PROGRAM Programma_2
VAR
    currentPlayer: BOOL;  // Bepaalt welke speler aan de beurt is
	zetGedaan: BOOL;
END_VAR

// Task 2: Speler zet zijn figuur
IF GVL.game_status = 1 THEN
    zetGedaan := FALSE; // Variabele om bij te houden of er een zet is gedaan

    // Bepaal welke speler aan de beurt is
    IF GVL.Player_1 THEN
        currentPlayer := TRUE;   // Speler 1 is actief
    ELSE
        currentPlayer := FALSE;  // Speler 2 is actief
    END_IF

    // Controleer of een rechthoek is geselecteerd en of deze leeg is
    // Als de rechthoek leeg is, vul het met het figuur van de speler
    IF GVL.Rechthoek_1 AND NOT (GVL.Driehoek_1 OR GVL.Rondje_1) THEN
        IF currentPlayer THEN
            GVL.Driehoek_1 := TRUE;  // Zet driehoek van speler 1
        ELSE
            GVL.Rondje_1 := TRUE;    // Zet rondje van speler 2
        END_IF
        zetGedaan := TRUE;
    ELSIF GVL.Rechthoek_2 AND NOT (GVL.Driehoek_2 OR GVL.Rondje_2) THEN
        IF currentPlayer THEN
            GVL.Driehoek_2 := TRUE;  // Zet driehoek van speler 1
        ELSE
            GVL.Rondje_2 := TRUE;    // Zet rondje van speler 2
        END_IF
        zetGedaan := TRUE;
    ELSIF GVL.Rechthoek_3 AND NOT (GVL.Driehoek_3 OR GVL.Rondje_3) THEN
        IF currentPlayer THEN
            GVL.Driehoek_3 := TRUE;  // Zet driehoek van speler 1
        ELSE
            GVL.Rondje_3 := TRUE;    // Zet rondje van speler 2
        END_IF
        zetGedaan := TRUE;
    ELSIF GVL.Rechthoek_4 AND NOT (GVL.Driehoek_4 OR GVL.Rondje_4) THEN
        IF currentPlayer THEN
            GVL.Driehoek_4 := TRUE;  // Zet driehoek van speler 1
        ELSE
            GVL.Rondje_4 := TRUE;    // Zet rondje van speler 2
        END_IF
        zetGedaan := TRUE;
    ELSIF GVL.Rechthoek_5 AND NOT (GVL.Driehoek_5 OR GVL.Rondje_5) THEN
        IF currentPlayer THEN
            GVL.Driehoek_5 := TRUE;  // Zet driehoek van speler 1
        ELSE
            GVL.Rondje_5 := TRUE;    // Zet rondje van speler 2
        END_IF
        zetGedaan := TRUE;
    ELSIF GVL.Rechthoek_6 AND NOT (GVL.Driehoek_6 OR GVL.Rondje_6) THEN
        IF currentPlayer THEN
            GVL.Driehoek_6 := TRUE;  // Zet driehoek van speler 1
        ELSE
            GVL.Rondje_6 := TRUE;    // Zet rondje van speler 2
        END_IF
        zetGedaan := TRUE;
    ELSIF GVL.Rechthoek_7 AND NOT (GVL.Driehoek_7 OR GVL.Rondje_7) THEN
        IF currentPlayer THEN
            GVL.Driehoek_7 := TRUE;  // Zet driehoek van speler 1
        ELSE
            GVL.Rondje_7 := TRUE;    // Zet rondje van speler 2
        END_IF
        zetGedaan := TRUE;
    ELSIF GVL.Rechthoek_8 AND NOT (GVL.Driehoek_8 OR GVL.Rondje_8) THEN
        IF currentPlayer THEN
            GVL.Driehoek_8 := TRUE;  // Zet driehoek van speler 1
        ELSE
            GVL.Rondje_8 := TRUE;    // Zet rondje van speler 2
        END_IF
        zetGedaan := TRUE;
    ELSIF GVL.Rechthoek_9 AND NOT (GVL.Driehoek_9 OR GVL.Rondje_9) THEN
        IF currentPlayer THEN
            GVL.Driehoek_9 := TRUE;  // Zet driehoek van speler 1
        ELSE
            GVL.Rondje_9 := TRUE;    // Zet rondje van speler 2
        END_IF
        zetGedaan := TRUE;
    END_IF

    // Wissel de beurt alleen als er een zet is gedaan en geen winnaar is
    IF zetGedaan AND GVL.winnaar = 0 THEN
        IF GVL.Player_1 THEN
            GVL.Player_1 := FALSE;   // Zet speler 1 uit
            GVL.Player_2 := TRUE;    // Zet speler 2 aan
            GVL.Player_1_Lamp := FALSE;  // Zet lamp van speler 1 uit
            GVL.Player_2_Lamp := TRUE;   // Zet lamp van speler 2 aan
        ELSE
            GVL.Player_1 := TRUE;    // Zet speler 1 aan
            GVL.Player_2 := FALSE;   // Zet speler 2 uit
            GVL.Player_1_Lamp := TRUE;  // Zet lamp van speler 1 aan
            GVL.Player_2_Lamp := FALSE;  // Zet lamp van speler 2 uit
        END_IF

        // Zet de status van het spel naar 2 (wincheck fase) als er een zet is gedaan
        GVL.game_status := 2;  // Ga naar de wincheck fase
    END_IF
END_IF

END_PROGRAM

(* stored: Version 1.1.0.1, ProductVersion 3.1.4024.12
   POU Programma_2: Id {ccfc2342-ac26-4787-a6a4-498199d0b244}, SpecialFunc None *)
